FUNCTION_BLOCK FB_HwRefTripleTrigger EXTENDS FB_CanNodeBase
VAR_INPUT
END_VAR
VAR_OUTPUT
END_VAR
VAR
	//PDOs
	nState 			AT %I* : ARRAY[1..3] OF USINT;
	nError 			AT %I* : USINT;
	nPeriod 		AT %Q* : ARRAY[1..3] OF UINT;
	nPulse 			AT %Q* : ARRAY[1..3] OF UINT;
	nPulseNumber 	AT %Q* : ARRAY[1..3] OF UINT;
	nVoltage 		AT %Q* : ARRAY[1..3] OF UINT;
	nCtrl 			AT %Q* : ARRAY[1..3] OF USINT;
	
	//SDOs
	nFrequency 			: ARRAY[1..3] OF DINT;
	nAmplitudePercent 	: ARRAY[1..3] OF UINT;
END_VAR

IF bNodeEnabled THEN
	SUPER^();
END_IF

METHOD M_SetPulse
VAR_INPUT
	nChannel : USINT;
	nPulse : UINT;
END_VAR
THIS^.nPulse[nChannel] := nPulse;
END_METHOD

METHOD M_SetFrequency
VAR_INPUT
	nChannel : USINT;
	nFrequency : DINT;
END_VAR
IF nFrequency > 0 THEN
	THIS^.nFrequency[nChannel] := nFrequency;
	nPeriod[nChannel] := DINT_TO_UINT(1000000 / nFrequency);
ELSE
	nPeriod[nChannel] := 0;
	THIS^.nFrequency[nChannel] := 0;
END_IF
END_METHOD

METHOD M_TriggerOn
VAR_INPUT
	nChannel : USINT;
	nPulseNumber : UINT;
END_VAR
THIS^.nPulseNumber[nChannel] := nPulseNumber;
nCtrl[nChannel] := 1;
END_METHOD

METHOD M_GetAmlitudeVolt : UINT
VAR_INPUT
	nChannel : USINT;
END_VAR
M_GetAmlitudeVolt := nVoltage[nChannel];
END_METHOD

METHOD M_TriggerOff
VAR_INPUT
	nChannel : USINT;
END_VAR
nCtrl[nChannel] := 0;
END_METHOD

METHOD M_GetState : BOOL
VAR_INPUT
	nChannel : USINT;
END_VAR
M_GetState := nState[nChannel].0;
END_METHOD

METHOD M_GetPulse : UINT
VAR_INPUT
	nChannel : USINT;
END_VAR
M_GetPulse := nPulse[nChannel];
END_METHOD

METHOD M_GetAmplitudePercent : UINT
VAR_INPUT
	nChannel : USINT;
END_VAR
M_GetAmplitudePercent := nAmplitudePercent[nChannel];
END_METHOD

METHOD M_SetAmplitudeVolt
VAR_INPUT
	nChannel : USINT;
	nValue : UINT;
END_VAR
nVoltage[nChannel] := LIMIT(0,nValue,10000);
nAmplitudePercent[nChannel] := nVoltage[nChannel] * 1000 / 10000;
END_METHOD

METHOD M_SetAmplitudePercent
VAR_INPUT
	nChannel : USINT;
	nValue : UINT;	//Zehntel %
END_VAR
nAmplitudePercent[nChannel] := LIMIT(0,nValue,1000);
nVoltage[nChannel] := 10000 / 1000 * nAmplitudePercent[nChannel];
END_METHOD

METHOD M_GetFrequency : DINT
VAR_INPUT
	nChannel : USINT;
END_VAR
M_GetFrequency := nFrequency[nChannel];
END_METHOD

END_FUNCTION_BLOCK

(* stored: Version 1.1.0.1, ProductVersion 3.1.0.25
   POU FB_HwRefTripleTrigger: Id {26cee8e2-36d9-4e41-bc0a-fec1b2da8863}
   Method M_SetPulse: Id {0bec5832-8e9e-4505-9c81-2655528a436b}
   Method M_SetFrequency: Id {15c430fe-87d5-4cb6-bfce-4fd5e98a425c}
   Method M_TriggerOn: Id {2ba45212-773c-419f-a142-57023ff6e62e}
   Method M_GetAmlitudeVolt: Id {339a69c5-feee-4259-9b1b-676e07a3a853}
   Method M_TriggerOff: Id {427320c8-9eaf-4a0d-be88-f5601914bbe4}
   Method M_GetState: Id {42971dd1-b7d4-4340-9ab1-5a7471b5c267}
   Method M_GetPulse: Id {91faeae8-62e1-4cb8-a967-cb4b0db0f46c}
   Method M_GetAmplitudePercent: Id {aaed8dbb-ba72-4034-ba37-74cd9daa3be1}
   Method M_SetAmplitudeVolt: Id {ab8a24c2-7675-4de9-85f8-9fc601f3f51c}
   Method M_SetAmplitudePercent: Id {b412a503-a1aa-4bf0-afb6-a3cc34bccead}
   Method M_GetFrequency: Id {c8d6a827-5acb-484a-938c-083024fe5667} *)
